TYPE Print_IO_typ:
STRUCT
	Inputs	: Print_Inputs_typ;
	Outputs	: Print_Outputs_typ;
END_STRUCT
END_TYPE

(* stored: Version 1.1.0.1, ProductVersion 3.1.4024.12
   DUT Print_IO_typ: Id {a793954f-8371-0095-1260-b7771e29c26f} *)
